// TIA Portal V18 export
DATA_BLOCK "event For datalogging"   // DB216
{ S7_Optimized_Access := 'TRUE' }
VERSION : 0.1
// stored: AutoNumber false, DBAccessibleFromOPCUA true, IsOnlyStoredInLoadMemory false, IsRetainMemResEnabled false, IsWriteProtectedInAS false, MemoryReserve 100
   VAR
      "event number" : Int := 1;
      "event number Moved" : Int := 1;
      "trigger Datalogging on event change" : Bool := FALSE;
      "production completed" : String[25] := 'Production End';
      Metering_running : Bool;
      Function_String : Array[0..13] of String[25];
   END_VAR
BEGIN
   Function_String[1] := 'machine idle';
   Function_String[2] := 'metering program running';
   Function_String[3] := 'ratio Check running';
   Function_String[4] := 'metering shot running';
   Function_String[5] := 'metering cont. running';
   Function_String[6] := 'Pre run running';
   Function_String[7] := 'Flush running';
   Function_String[8] := 'Deaerate running';
   Function_String[9] := 'machine Faulty';
   Function_String[10] := 'emergency stop';
   Function_String[11] := 'regenration running';
   Function_String[12] := 'dosing completed';
END_DATA_BLOCK
